// TIA Portal V16 export
// export: Created 2022-02-11T14:39:21.4185203Z, ExportSetting WithDefaults, DisplayName Totally Integrated Automation Portal, DisplayVersion V16 Update 1, DisplayName TIA Portal Version Control Interface, DisplayVersion V16, DisplayName TIA Portal Openness, DisplayVersion V16, DisplayName SINAMICS Startdrive Advanced, DisplayVersion V16 Update 5, DisplayName SINAMICS Startdrive G130, G150, S120, S150, SINAMICS MV, S210, DisplayVersion V16 Update 5, DisplayName SINAMICS Startdrive G110M, G120, G120C, G120D, G120P, G115D, DisplayVersion V16 Update 5, DisplayName STEP 7 Professional, DisplayVersion V16, DisplayName STEP 7 Safety, DisplayVersion V16, DisplayName WinCC Advanced, DisplayVersion V16, DisplayName SIMATIC Visualization Architect, DisplayVersion V16
DATA_BLOCK "ПФМ Брака_DB"   // DB8
VERSION : 0.1
// stored: AutoNumber true, InstanceOfName ПФМ Брака, InstanceOfType FB
"ПФМ Брака"
   // VAR RETAIN
   //    Trig332 : Bool;
   //    "TrigS79.3" : Bool;
   //    ForcingPacket : Bool;
   //    LiftPushingPacket : Bool;
   //    HodVil2 { ExternalAccessible := 'False'; ExternalVisible := 'False'; ExternalWritable := 'False'} : Bool;
   //    HodVil { ExternalAccessible := 'False'; ExternalVisible := 'False'; ExternalWritable := 'False'} : Bool;
   //    ForcingLift : Bool;
   //    CountSensor_front : Bool;
   //    StopDovod : Bool;
   //    StopDropppingBoards : Bool;
   //    newBob_old : Bool;
   //    liftDown_old : Bool;
   //    liftPushingPacket_old : Bool;
   //    newBoard_old : Bool;
   //    Upor_Off_trig : Bool;
   //    Lift_GoToStartPosition : Bool;
   //    ReviveSignal : Bool;
   //    StartAwaitForGasket : Bool;
   //    AwaitGasket : Bool;
   //    AlarmNotReadedPack : Bool;
   //    AlarmExtraBoardInLay : Bool;
   //    AlarmNoPacketPushed : Bool;
   //    BoardsInLayCounter : Int;
   //    LayersCounter : Int;
   //    Board_counter : "Adder";
   //    Lay_counter : "Adder";
   // END_VAR
BEGIN
END_DATA_BLOCK
